FUNCTION_BLOCK TEST_CAST (* Regression Test  of type casting in ST replacement *)
  (* Standard: 61499-2 *)
  (* Version 0.1, 2006-09-06, JHC, JHC, Made a SimpleFB *)
  (* Version 0.0, 2002-12-17, JHC, Rockwell Automation *)
  (* Compiler header: package fb.rt.test; *)
  (* Compiler classdef: SimpleFB *)
  (* Compiler Java Sun JDK 1.5.0 *)
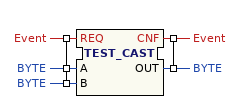
  EVENT_INPUT
    REQ WITH A, B; (* Normal Execution Request *)
  END_EVENT
  EVENT_OUTPUT
    CNF WITH OUT; (* Execution Confirmation *)
  END_EVENT
  VAR_INPUT
    A : BYTE;
    B : BYTE;
  END_VAR
  VAR_OUTPUT
    OUT : BYTE; (* A & B? *)
  END_VAR
  ALGORITHM REQ IN ST: (* Normally executed algorithm *)
OUT := A & B;
  END_ALGORITHM
END_FUNCTION_BLOCK
